# EPICS substitutions: sans2dApertureWaveguidesApp/Db/sans2d_apertures_waveguides.substitutions
global {P=\$(P),MYPVPREFIX=\$(MYPVPREFIX)}

file "$(TOP)/sans2dApertureWaveguidesApp/Db/stop_motion.template" {
	{FULL_PREFIX="\$(P)SANS2DAPWV:"}
}

file "$(TOP)/sans2dApertureWaveguidesApp/Db/inhibit_motion.template" {
	{FULL_PREFIX="\$(P)SANS2DAPWV:"}
}

file "$(TOP)/sans2dApertureWaveguidesApp/Db/positional_error.template" {
	pattern {P ,M}
    {"\$(P)", "MTR\$(CCP_01)01"}
    {"\$(P)", "MTR\$(CCP_01)02"}
    {"\$(P)", "MTR\$(CCP_01)03"}
    {"\$(P)", "MTR\$(CCP_01)04"}
    {"\$(P)", "MTR\$(CCP_01)05"}

    {"\$(P)", "MTR\$(CCP_02)01"}
    {"\$(P)", "MTR\$(CCP_02)02"}
    {"\$(P)", "MTR\$(CCP_02)03"}
    {"\$(P)", "MTR\$(CCP_02)04"}
    {"\$(P)", "MTR\$(CCP_02)05"}
}
